    // Event "Pumpcellars_MiddlePumpcellar_Mode_c_off".
    IF NOT progress THEN
        b2 := (state0.dvar_M_Pumpcellars_MiddlePumpcellar_Mode) = (elit_drain);
        b2 := b2 OR ((state0.dvar_M_Pumpcellars_MiddlePumpcellar_Mode) = (elit_store));
        b1 := b2;
        b1 := b1 AND ((state0.dvar_M_RequirementStateEvtExcls) = (elit_X));
        IF b1 THEN
            b2 := (state0.dvar_M_Pumpcellars_MiddlePumpcellar_Control_Observer) = (elit_unpressed);
            IF NOT(b2) THEN
                b3 := (state0.dvar_M_Pumpcellars_MiddlePumpcellar_Control_Mode) = (elit_manual);
                b3 := b3 AND ((state0.dvar_M_Pumpcellars_MiddlePumpcellar_Control_Observer) <> (elit_autoPressed));
                b2 := b2 OR (b3);
            END_IF;
            b1 := b1 AND (b2);
        END_IF;
        b1 := b1 AND ((state0.dvar_M_Pumpcellars_MiddlePumpcellar_Control_Mode) = (elit_manual));
        b1 := b1 AND ((state0.dvar_M_Pumpcellars_MiddlePumpcellar_Control_Observer) = (elit_offPressed));
        b1 := b1 AND ((state0.dvar_M_Mutex1Home_TokenTracker) = (elit_Home));
        b1 := b1 AND ((state0.dvar_M_Mutex2Home_TokenTracker) = (elit_Home));
        b1 := b1 AND ((state0.dvar_M_sup1a) = (elit_X));
        b1 := b1 AND ((state0.dvar_M_sup2) = (elit_X));
        b1 := b1 AND ((state0.dvar_M_sup4) = (elit_X));
        IF b1 THEN
            progress := TRUE;
            state1 := state0;

            IF ((state0.dvar_M_HWMPCMode) = (elit_drain)) THEN
                state1.dvar_M_HWMPCMode_DRAIN := FALSE;
                state1.dvar_M_HWMPCMode_STORE := FALSE;
                state1.dvar_M_HWMPCMode_OFF := TRUE;
                state1.dvar_M_HWMPCMode := elit_off;
            ELSIF ((state0.dvar_M_HWMPCMode) = (elit_store)) THEN
                state1.dvar_M_HWMPCMode_DRAIN := FALSE;
                state1.dvar_M_HWMPCMode_STORE := FALSE;
                state1.dvar_M_HWMPCMode_OFF := TRUE;
                state1.dvar_M_HWMPCMode := elit_off;
            ELSIF ((state0.dvar_M_HWMPCMode) = (elit_off)) THEN
                state1.dvar_M_HWMPCMode := elit_off;
            END_IF;
            IF ((state0.dvar_M_Pumpcellars_MiddlePumpcellar_Mode) = (elit_drain)) THEN
                state1.dvar_M_Pumpcellars_MiddlePumpcellar_Mode := elit_off;
            ELSIF ((state0.dvar_M_Pumpcellars_MiddlePumpcellar_Mode) = (elit_store)) THEN
                state1.dvar_M_Pumpcellars_MiddlePumpcellar_Mode := elit_off;
            END_IF;

            state0 := state1;
        END_IF;
    END_IF;

    // Event "Pumpcellars_MiddlePumpcellar_Mode_c_store".
    IF NOT progress THEN
        b2 := (state0.dvar_M_Pumpcellars_MiddlePumpcellar_Mode) = (elit_drain);
        b2 := b2 OR ((state0.dvar_M_Pumpcellars_MiddlePumpcellar_Mode) = (elit_off));
        b1 := b2;
        b1 := b1 AND ((state0.dvar_M_RequirementStateEvtExcls) = (elit_X));
        IF b1 THEN
            b2 := (state0.dvar_M_Pumpcellars_MiddlePumpcellar_Control_Observer) = (elit_unpressed);
            IF NOT(b2) THEN
                b3 := (state0.dvar_M_Pumpcellars_MiddlePumpcellar_Control_Mode) = (elit_manual);
                b3 := b3 AND ((state0.dvar_M_Pumpcellars_MiddlePumpcellar_Control_Observer) <> (elit_autoPressed));
                b2 := b2 OR (b3);
            END_IF;
            b1 := b1 AND (b2);
        END_IF;
        IF b1 THEN
            b3 := (state0.dvar_M_Pumpcellars_MiddlePumpcellar_Control_Mode) = (elit_auto);
            b3 := b3 AND (NOT(((state0.dvar_M_Pumpcellars_Traffictube1_ModeTraffictube_Observer) = (elit_operational)) AND ((state0.dvar_M_Pumpcellars_Traffictube2_ModeTraffictube_Observer) = (elit_operational))));
            b2 := b3;
            IF NOT(b2) THEN
                b3 := (state0.dvar_M_Pumpcellars_MiddlePumpcellar_Control_Mode) = (elit_manual);
                b3 := b3 AND ((state0.dvar_M_Pumpcellars_MiddlePumpcellar_Control_Observer) = (elit_storePressed));
                b2 := b2 OR (b3);
            END_IF;
            b1 := b1 AND (b2);
        END_IF;
        b1 := b1 AND ((state0.dvar_M_Mutex1Home_TokenTracker) = (elit_Home));
        b1 := b1 AND ((state0.dvar_M_Mutex2Home_TokenTracker) = (elit_Home));
        b1 := b1 AND ((state0.dvar_M_sup1a) = (elit_X));
        b1 := b1 AND ((state0.dvar_M_sup2) = (elit_X));
        b1 := b1 AND ((state0.dvar_M_sup4) = (elit_X));
        IF b1 THEN
            progress := TRUE;
            state1 := state0;

            IF ((state0.dvar_M_HWMPCMode) = (elit_drain)) THEN
                state1.dvar_M_HWMPCMode_DRAIN := FALSE;
                state1.dvar_M_HWMPCMode_STORE := TRUE;
                state1.dvar_M_HWMPCMode_OFF := FALSE;
                state1.dvar_M_HWMPCMode := elit_store;
            ELSIF ((state0.dvar_M_HWMPCMode) = (elit_store)) THEN
                state1.dvar_M_HWMPCMode := elit_store;
            ELSIF ((state0.dvar_M_HWMPCMode) = (elit_off)) THEN
                state1.dvar_M_HWMPCMode_DRAIN := FALSE;
                state1.dvar_M_HWMPCMode_STORE := TRUE;
                state1.dvar_M_HWMPCMode_OFF := FALSE;
                state1.dvar_M_HWMPCMode := elit_store;
            END_IF;
            IF ((state0.dvar_M_Pumpcellars_MiddlePumpcellar_Mode) = (elit_drain)) THEN
                state1.dvar_M_Pumpcellars_MiddlePumpcellar_Mode := elit_store;
            ELSIF ((state0.dvar_M_Pumpcellars_MiddlePumpcellar_Mode) = (elit_off)) THEN
                state1.dvar_M_Pumpcellars_MiddlePumpcellar_Mode := elit_store;
            END_IF;

            state0 := state1;
        END_IF;
    END_IF;

    // Event "Pumpcellars_MiddlePumpcellar_PompRichting_c_hoofdPumpcellars1".
    IF NOT progress THEN
        IF (state0.dvar_M_MPC_HWPomprichting) = (elit_X) THEN
            progress := TRUE;
            state1 := state0;

            state1.dvar_M_MPC_HWPomprichting_HPC1 := TRUE;

            state0 := state1;
        END_IF;
    END_IF;

    // Event "Pumpcellars_MiddlePumpcellar_PompRichting_c_hoofdPumpcellars2".
    IF NOT progress THEN
        IF (state0.dvar_M_MPC_HWPomprichting) = (elit_X) THEN
            progress := TRUE;
            state1 := state0;

            state1.dvar_M_MPC_HWPomprichting_HPC1 := FALSE;

            state0 := state1;
        END_IF;
    END_IF;

    // Event "Pumpcellars_MiddlePumpcellar_Pump1_c_off".
    IF NOT progress THEN
        b1 := (state0.dvar_M_MPC_HWPump1) = (elit_X);
        b1 := b1 AND ((state0.dvar_M_Pumpcellars_MiddlePumpcellar_Pump1) = (elit_on));
        b1 := b1 AND ((state0.dvar_M_RequirementStateEvtExcls) = (elit_X));
        IF b1 THEN
            b3 := (state0.dvar_M_Pumpcellars_MiddlePumpcellar_Mode) = (elit_store);
            IF b3 THEN
                b4 := (state0.dvar_M_Pumpcellars_MiddlePumpcellar_SensorTank) = (elit_S2);
                b4 := b4 OR ((state0.dvar_M_Pumpcellars_MiddlePumpcellar_SensorTank) = (elit_S3));
                b4 := b4 OR ((state0.dvar_M_Pumpcellars_MiddlePumpcellar_SensorTank) = (elit_S1));
                b4 := b4 OR ((state0.dvar_M_Pumpcellars_MiddlePumpcellar_SensorTank) = (elit_Empty));
                b3 := b3 AND (b4);
            END_IF;
            b2 := b3;
            IF NOT(b2) THEN
                b3 := (state0.dvar_M_Pumpcellars_MiddlePumpcellar_Mode) = (elit_drain);
                b3 := b3 AND ((state0.dvar_M_Pumpcellars_MiddlePumpcellar_SensorTank) = (elit_Empty));
                b2 := b2 OR (b3);
            END_IF;
            b2 := b2 OR ((state0.dvar_M_Pumpcellars_MiddlePumpcellar_Mode) = (elit_off));
            b1 := b1 AND (b2);
        END_IF;
        b1 := b1 AND ((state0.dvar_M_Pumpcellars_MiddlePumpcellar_Control_Observer) = (elit_unpressed));
        b1 := b1 AND ((state0.dvar_M_sup2) = (elit_X));
        IF b1 THEN
            progress := TRUE;
            state1 := state0;

            state1.dvar_M_MPC_HWPump1_ON := FALSE;
            state1.dvar_M_Pumpcellars_MiddlePumpcellar_Pump1 := elit_off;

            state0 := state1;
        END_IF;
    END_IF;

    // Event "Pumpcellars_MiddlePumpcellar_Pump1_c_on".
    IF NOT progress THEN
        b1 := (state0.dvar_M_MPC_HWPump1) = (elit_X);
        b1 := b1 AND ((state0.dvar_M_Pumpcellars_MiddlePumpcellar_Pump1) = (elit_off));
        b1 := b1 AND ((state0.dvar_M_RequirementStateEvtExcls) = (elit_X));
        IF b1 THEN
            b3 := (state0.dvar_M_Pumpcellars_MiddlePumpcellar_Mode) = (elit_store);
            b3 := b3 AND ((state0.dvar_M_Pumpcellars_MiddlePumpcellar_SensorTank) = (elit_S5));
            b2 := b3;
            IF NOT(b2) THEN
                b3 := (state0.dvar_M_Pumpcellars_MiddlePumpcellar_Mode) = (elit_drain);
                IF b3 THEN
                    b4 := (state0.dvar_M_Pumpcellars_MiddlePumpcellar_SensorTank) = (elit_S2);
                    b4 := b4 OR ((state0.dvar_M_Pumpcellars_MiddlePumpcellar_SensorTank) = (elit_S3));
                    b4 := b4 OR ((state0.dvar_M_Pumpcellars_MiddlePumpcellar_SensorTank) = (elit_S4));
                    b4 := b4 OR ((state0.dvar_M_Pumpcellars_MiddlePumpcellar_SensorTank) = (elit_S5));
                    b3 := b3 AND (b4);
                END_IF;
                b2 := b2 OR (b3);
            END_IF;
            b1 := b1 AND (b2);
        END_IF;
        b1 := b1 AND ((state0.dvar_M_Pumpcellars_MiddlePumpcellar_Control_Observer) = (elit_unpressed));
        b1 := b1 AND ((state0.dvar_M_sup2) = (elit_X));
        IF b1 THEN
            progress := TRUE;
            state1 := state0;

            state1.dvar_M_MPC_HWPump1_ON := TRUE;
            state1.dvar_M_Pumpcellars_MiddlePumpcellar_Pump1 := elit_on;

            state0 := state1;
        END_IF;
    END_IF;

    // Event "Pumpcellars_MiddlePumpcellar_Pump2_c_off".
    IF NOT progress THEN
        b1 := (state0.dvar_M_MPC_HWPump2) = (elit_X);
        b1 := b1 AND ((state0.dvar_M_Pumpcellars_MiddlePumpcellar_Pump2) = (elit_on));
        b1 := b1 AND ((state0.dvar_M_RequirementStateEvtExcls) = (elit_X));
        IF b1 THEN
            b3 := (state0.dvar_M_Pumpcellars_MiddlePumpcellar_Mode) = (elit_store);
            IF b3 THEN
                b4 := (state0.dvar_M_Pumpcellars_MiddlePumpcellar_SensorTank) = (elit_S2);
                b4 := b4 OR ((state0.dvar_M_Pumpcellars_MiddlePumpcellar_SensorTank) = (elit_S3));
                b4 := b4 OR ((state0.dvar_M_Pumpcellars_MiddlePumpcellar_SensorTank) = (elit_S1));
                b4 := b4 OR ((state0.dvar_M_Pumpcellars_MiddlePumpcellar_SensorTank) = (elit_Empty));
                b3 := b3 AND (b4);
            END_IF;
            b2 := b3;
            IF NOT(b2) THEN
                b3 := (state0.dvar_M_Pumpcellars_MiddlePumpcellar_Mode) = (elit_drain);
                b3 := b3 AND ((state0.dvar_M_Pumpcellars_MiddlePumpcellar_SensorTank) = (elit_Empty));
                b2 := b2 OR (b3);
            END_IF;
            b2 := b2 OR ((state0.dvar_M_Pumpcellars_MiddlePumpcellar_Mode) = (elit_off));
            b1 := b1 AND (b2);
        END_IF;
        b1 := b1 AND ((state0.dvar_M_Pumpcellars_MiddlePumpcellar_Control_Observer) = (elit_unpressed));
        b1 := b1 AND ((state0.dvar_M_sup2) = (elit_X));
        IF b1 THEN
            progress := TRUE;
            state1 := state0;

            state1.dvar_M_MPC_HWPump2_ON := FALSE;
            state1.dvar_M_Pumpcellars_MiddlePumpcellar_Pump2 := elit_off;

            state0 := state1;
        END_IF;
    END_IF;

    // Event "Pumpcellars_MiddlePumpcellar_Pump2_c_on".
    IF NOT progress THEN
        b1 := (state0.dvar_M_MPC_HWPump2) = (elit_X);
        b1 := b1 AND ((state0.dvar_M_Pumpcellars_MiddlePumpcellar_Pump2) = (elit_off));
        b1 := b1 AND ((state0.dvar_M_RequirementStateEvtExcls) = (elit_X));
        IF b1 THEN
            b3 := (state0.dvar_M_Pumpcellars_MiddlePumpcellar_Mode) = (elit_store);
            b3 := b3 AND ((state0.dvar_M_Pumpcellars_MiddlePumpcellar_SensorTank) = (elit_S5));
            b2 := b3;
            IF NOT(b2) THEN
                b3 := (state0.dvar_M_Pumpcellars_MiddlePumpcellar_Mode) = (elit_drain);
                IF b3 THEN
                    b4 := (state0.dvar_M_Pumpcellars_MiddlePumpcellar_SensorTank) = (elit_S3);
                    b4 := b4 OR ((state0.dvar_M_Pumpcellars_MiddlePumpcellar_SensorTank) = (elit_S4));
                    b4 := b4 OR ((state0.dvar_M_Pumpcellars_MiddlePumpcellar_SensorTank) = (elit_S5));
                    b3 := b3 AND (b4);
                END_IF;
                b2 := b2 OR (b3);
            END_IF;
            b1 := b1 AND (b2);
        END_IF;
        b1 := b1 AND ((state0.dvar_M_Pumpcellars_MiddlePumpcellar_Control_Observer) = (elit_unpressed));
        b1 := b1 AND ((state0.dvar_M_sup2) = (elit_X));
        IF b1 THEN
            progress := TRUE;
            state1 := state0;

            state1.dvar_M_MPC_HWPump2_ON := TRUE;
            state1.dvar_M_Pumpcellars_MiddlePumpcellar_Pump2 := elit_on;

            state0 := state1;
        END_IF;
    END_IF;

    // Event "Pumpcellars_MiddlePumpcellar_PumpDirection_c_headPumpcellar1".
    IF NOT progress THEN
        b1 := (state0.dvar_M_Pumpcellars_MiddlePumpcellar_PumpDirection) = (elit_headPumpcellar2);
        b1 := b1 AND ((state0.dvar_M_RequirementStateEvtExcls) = (elit_X));
        b1 := b1 AND ((state0.dvar_M_Pumpcellars_HeadPumpcellar1_SensorTank) = (elit_S4));
        b1 := b1 AND ((state0.dvar_M_sup5) = (elit_X));
        IF b1 THEN
            progress := TRUE;
            state1 := state0;

            state1.dvar_M_Pumpcellars_MiddlePumpcellar_PumpDirection := elit_headPumpcellar1;

            state0 := state1;
        END_IF;
    END_IF;

    // Event "Pumpcellars_MiddlePumpcellar_PumpDirection_c_headPumpcellar2".
    IF NOT progress THEN
        b1 := (state0.dvar_M_Pumpcellars_MiddlePumpcellar_PumpDirection) = (elit_headPumpcellar1);
        b1 := b1 AND ((state0.dvar_M_RequirementStateEvtExcls) = (elit_X));
        b1 := b1 AND ((state0.dvar_M_Pumpcellars_HeadPumpcellar1_SensorTank) = (elit_S5));
        b1 := b1 AND ((state0.dvar_M_sup5) = (elit_X));
        IF b1 THEN
            progress := TRUE;
            state1 := state0;

            state1.dvar_M_Pumpcellars_MiddlePumpcellar_PumpDirection := elit_headPumpcellar2;

            state0 := state1;
        END_IF;
    END_IF;

    // Event "Pumpcellars_MiddlePumpcellar_SensorTank_u_S1off".
    IF NOT progress THEN
        b1 := (state0.dvar_M_MPC_HWSensorS1) = (elit_on);
        b1 := b1 AND (NOT(ivar_M_MPC_HWSensorS1_ON));
        b1 := b1 AND ((state0.dvar_M_Pumpcellars_MiddlePumpcellar_SensorTank) = (elit_S1));
        IF b1 THEN
            b2 := (state0.dvar_M_Pumpcellars_MiddlePumpcellar_Pump1) = (elit_on);
            b2 := b2 OR ((state0.dvar_M_Pumpcellars_MiddlePumpcellar_Pump2) = (elit_on));
            b1 := b1 AND (b2);
        END_IF;
        IF b1 THEN
            progress := TRUE;
            state1 := state0;

            state1.dvar_M_MPC_HWSensorS1 := elit_off;
            state1.dvar_M_Pumpcellars_MiddlePumpcellar_SensorTank := elit_Empty;

            state0 := state1;
        END_IF;
    END_IF;

    // Event "Pumpcellars_MiddlePumpcellar_SensorTank_u_S1on".
    IF NOT progress THEN
        b1 := (state0.dvar_M_MPC_HWSensorS1) = (elit_off);
        b1 := b1 AND (ivar_M_MPC_HWSensorS1_ON);
        b1 := b1 AND ((state0.dvar_M_Pumpcellars_MiddlePumpcellar_SensorTank) = (elit_Empty));
        IF b1 THEN
            progress := TRUE;
            state1 := state0;

            state1.dvar_M_MPC_HWSensorS1 := elit_on;
            state1.dvar_M_Pumpcellars_MiddlePumpcellar_SensorTank := elit_S1;

            state0 := state1;
        END_IF;
    END_IF;

    // Event "Pumpcellars_MiddlePumpcellar_SensorTank_u_S2off".
    IF NOT progress THEN
        b1 := (state0.dvar_M_MPC_HWSensorS2) = (elit_on);
        b1 := b1 AND (NOT(ivar_M_MPC_HWSensorS2_ON));
        b1 := b1 AND ((state0.dvar_M_Pumpcellars_MiddlePumpcellar_SensorTank) = (elit_S2));
        IF b1 THEN
            b2 := (state0.dvar_M_Pumpcellars_MiddlePumpcellar_Pump1) = (elit_on);
            b2 := b2 OR ((state0.dvar_M_Pumpcellars_MiddlePumpcellar_Pump2) = (elit_on));
            b1 := b1 AND (b2);
        END_IF;
        IF b1 THEN
            progress := TRUE;
            state1 := state0;

            state1.dvar_M_MPC_HWSensorS2 := elit_off;
            state1.dvar_M_Pumpcellars_MiddlePumpcellar_SensorTank := elit_S1;

            state0 := state1;
        END_IF;
    END_IF;

    // Event "Pumpcellars_MiddlePumpcellar_SensorTank_u_S2on".
    IF NOT progress THEN
        b1 := (state0.dvar_M_MPC_HWSensorS2) = (elit_off);
        b1 := b1 AND (ivar_M_MPC_HWSensorS2_ON);
        b1 := b1 AND ((state0.dvar_M_Pumpcellars_MiddlePumpcellar_SensorTank) = (elit_S1));
        IF b1 THEN
            progress := TRUE;
            state1 := state0;

            state1.dvar_M_MPC_HWSensorS2 := elit_on;
            state1.dvar_M_Pumpcellars_MiddlePumpcellar_SensorTank := elit_S2;

            state0 := state1;
        END_IF;
    END_IF;

    // Event "Pumpcellars_MiddlePumpcellar_SensorTank_u_S3off".
    IF NOT progress THEN
        b1 := (state0.dvar_M_MPC_HWSensorS3) = (elit_on);
        b1 := b1 AND (NOT(ivar_M_MPC_HWSensorS3_ON));
        b1 := b1 AND ((state0.dvar_M_Pumpcellars_MiddlePumpcellar_SensorTank) = (elit_S3));
        IF b1 THEN
            b2 := (state0.dvar_M_Pumpcellars_MiddlePumpcellar_Pump1) = (elit_on);
            b2 := b2 OR ((state0.dvar_M_Pumpcellars_MiddlePumpcellar_Pump2) = (elit_on));
            b1 := b1 AND (b2);
        END_IF;
        IF b1 THEN
            progress := TRUE;
            state1 := state0;

            state1.dvar_M_MPC_HWSensorS3 := elit_off;
            state1.dvar_M_Pumpcellars_MiddlePumpcellar_SensorTank := elit_S2;

            state0 := state1;
        END_IF;
    END_IF;

    // Event "Pumpcellars_MiddlePumpcellar_SensorTank_u_S3on".
    IF NOT progress THEN
        b1 := (state0.dvar_M_MPC_HWSensorS3) = (elit_off);
        b1 := b1 AND (ivar_M_MPC_HWSensorS3_ON);
        b1 := b1 AND ((state0.dvar_M_Pumpcellars_MiddlePumpcellar_SensorTank) = (elit_S2));
        IF b1 THEN
            progress := TRUE;
            state1 := state0;

            state1.dvar_M_MPC_HWSensorS3 := elit_on;
            state1.dvar_M_Pumpcellars_MiddlePumpcellar_SensorTank := elit_S3;

            state0 := state1;
        END_IF;
    END_IF;

    // Event "Pumpcellars_MiddlePumpcellar_SensorTank_u_S4off".
    IF NOT progress THEN
        b1 := (state0.dvar_M_MPC_HWSensorS4) = (elit_on);
        b1 := b1 AND (NOT(ivar_M_MPC_HWSensorS4_ON));
        b1 := b1 AND ((state0.dvar_M_Pumpcellars_MiddlePumpcellar_SensorTank) = (elit_S4));
        IF b1 THEN
            b2 := (state0.dvar_M_Pumpcellars_MiddlePumpcellar_Pump1) = (elit_on);
            b2 := b2 OR ((state0.dvar_M_Pumpcellars_MiddlePumpcellar_Pump2) = (elit_on));
            b1 := b1 AND (b2);
        END_IF;
        IF b1 THEN
            progress := TRUE;
            state1 := state0;

            state1.dvar_M_MPC_HWSensorS4 := elit_off;
            state1.dvar_M_Pumpcellars_MiddlePumpcellar_SensorTank := elit_S3;

            state0 := state1;
        END_IF;
    END_IF;

    // Event "Pumpcellars_MiddlePumpcellar_SensorTank_u_S4on".
    IF NOT progress THEN
        b1 := (state0.dvar_M_MPC_HWSensorS4) = (elit_off);
        b1 := b1 AND (ivar_M_MPC_HWSensorS4_ON);
        b1 := b1 AND ((state0.dvar_M_Pumpcellars_MiddlePumpcellar_SensorTank) = (elit_S3));
        IF b1 THEN
            progress := TRUE;
            state1 := state0;

            state1.dvar_M_MPC_HWSensorS4 := elit_on;
            state1.dvar_M_Pumpcellars_MiddlePumpcellar_SensorTank := elit_S4;

            state0 := state1;
        END_IF;
    END_IF;

    // Event "Pumpcellars_MiddlePumpcellar_SensorTank_u_S5off".
    IF NOT progress THEN
        b1 := (state0.dvar_M_MPC_HWSensorS5) = (elit_on);
        b1 := b1 AND (NOT(ivar_M_MPC_HWSensorS5_ON));
        b1 := b1 AND ((state0.dvar_M_Pumpcellars_MiddlePumpcellar_SensorTank) = (elit_S5));
        IF b1 THEN
            b2 := (state0.dvar_M_Pumpcellars_MiddlePumpcellar_Pump1) = (elit_on);
            b2 := b2 OR ((state0.dvar_M_Pumpcellars_MiddlePumpcellar_Pump2) = (elit_on));
            b1 := b1 AND (b2);
        END_IF;
        IF b1 THEN
            progress := TRUE;
            state1 := state0;

            state1.dvar_M_MPC_HWSensorS5 := elit_off;
            state1.dvar_M_Pumpcellars_MiddlePumpcellar_SensorTank := elit_S4;

            state0 := state1;
        END_IF;
    END_IF;

    // Event "Pumpcellars_MiddlePumpcellar_SensorTank_u_S5on".
    IF NOT progress THEN
        b1 := (state0.dvar_M_MPC_HWSensorS5) = (elit_off);
        b1 := b1 AND (ivar_M_MPC_HWSensorS5_ON);
        b1 := b1 AND ((state0.dvar_M_Pumpcellars_MiddlePumpcellar_SensorTank) = (elit_S4));
        IF b1 THEN
            progress := TRUE;
            state1 := state0;

            state1.dvar_M_MPC_HWSensorS5 := elit_on;
            state1.dvar_M_Pumpcellars_MiddlePumpcellar_SensorTank := elit_S5;

            state0 := state1;
        END_IF;
    END_IF;

    // Event "Pumpcellars_Traffictube1_Observer_c_emergency".
    IF NOT progress THEN
        b1 := (state0.dvar_M_HWModeTraffictube1Observer) = (elit_X);
        b1 := b1 AND (ivar_TT1EMERGENCY);
        b1 := b1 AND (NOT(ivar_TT1OPERATIONAL));
        b1 := b1 AND (NOT(ivar_TT1RECOVERY));
        IF b1 THEN
            b2 := (state0.dvar_M_Pumpcellars_Traffictube1_ModeTraffictube_Observer) = (elit_operational);
            b2 := b2 OR ((state0.dvar_M_Pumpcellars_Traffictube1_ModeTraffictube_Observer) = (elit_recovery));
            b1 := b1 AND (b2);
        END_IF;
        IF b1 THEN
            progress := TRUE;
            state1 := state0;

            IF ((state0.dvar_M_Pumpcellars_Traffictube1_ModeTraffictube_Observer) = (elit_operational)) THEN
                state1.dvar_M_Pumpcellars_Traffictube1_ModeTraffictube_Observer := elit_emergency;
            ELSIF ((state0.dvar_M_Pumpcellars_Traffictube1_ModeTraffictube_Observer) = (elit_recovery)) THEN
                state1.dvar_M_Pumpcellars_Traffictube1_ModeTraffictube_Observer := elit_emergency;
            END_IF;

            state0 := state1;
        END_IF;
    END_IF;

    // Event "Pumpcellars_Traffictube1_Observer_c_operational".
    IF NOT progress THEN
        b1 := (state0.dvar_M_HWModeTraffictube1Observer) = (elit_X);
        b1 := b1 AND (NOT(ivar_TT1EMERGENCY));
        b1 := b1 AND (ivar_TT1OPERATIONAL);
        b1 := b1 AND (NOT(ivar_TT1RECOVERY));
        IF b1 THEN
            b2 := (state0.dvar_M_Pumpcellars_Traffictube1_ModeTraffictube_Observer) = (elit_emergency);
            b2 := b2 OR ((state0.dvar_M_Pumpcellars_Traffictube1_ModeTraffictube_Observer) = (elit_recovery));
            b1 := b1 AND (b2);
        END_IF;
        IF b1 THEN
            progress := TRUE;
            state1 := state0;

            IF ((state0.dvar_M_Pumpcellars_Traffictube1_ModeTraffictube_Observer) = (elit_emergency)) THEN
                state1.dvar_M_Pumpcellars_Traffictube1_ModeTraffictube_Observer := elit_operational;
            ELSIF ((state0.dvar_M_Pumpcellars_Traffictube1_ModeTraffictube_Observer) = (elit_recovery)) THEN
                state1.dvar_M_Pumpcellars_Traffictube1_ModeTraffictube_Observer := elit_operational;
            END_IF;

            state0 := state1;
        END_IF;
    END_IF;

    // Event "Pumpcellars_Traffictube1_Observer_c_recovery".
    IF NOT progress THEN
        b1 := (state0.dvar_M_HWModeTraffictube1Observer) = (elit_X);
        b1 := b1 AND (NOT(ivar_TT1EMERGENCY));
        b1 := b1 AND (NOT(ivar_TT1OPERATIONAL));
        b1 := b1 AND (ivar_TT1RECOVERY);
        IF b1 THEN
            b2 := (state0.dvar_M_Pumpcellars_Traffictube1_ModeTraffictube_Observer) = (elit_operational);
            b2 := b2 OR ((state0.dvar_M_Pumpcellars_Traffictube1_ModeTraffictube_Observer) = (elit_emergency));
            b1 := b1 AND (b2);
        END_IF;
        IF b1 THEN
            progress := TRUE;
            state1 := state0;

            IF ((state0.dvar_M_Pumpcellars_Traffictube1_ModeTraffictube_Observer) = (elit_operational)) THEN
                state1.dvar_M_Pumpcellars_Traffictube1_ModeTraffictube_Observer := elit_recovery;
            ELSIF ((state0.dvar_M_Pumpcellars_Traffictube1_ModeTraffictube_Observer) = (elit_emergency)) THEN
                state1.dvar_M_Pumpcellars_Traffictube1_ModeTraffictube_Observer := elit_recovery;
            END_IF;

            state0 := state1;
        END_IF;
    END_IF;

    // Event "Pumpcellars_Traffictube2_Observer_c_emergency".
    IF NOT progress THEN
        b1 := (state0.dvar_M_HWModeTraffictube2Observer) = (elit_X);
        b1 := b1 AND (ivar_TT2EMERGENCY);
        b1 := b1 AND (NOT(ivar_TT2OPERATIONAL));
        b1 := b1 AND (NOT(ivar_TT2RECOVERY));
        IF b1 THEN
            b2 := (state0.dvar_M_Pumpcellars_Traffictube2_ModeTraffictube_Observer) = (elit_operational);
            b2 := b2 OR ((state0.dvar_M_Pumpcellars_Traffictube2_ModeTraffictube_Observer) = (elit_recovery));
            b1 := b1 AND (b2);
        END_IF;
        IF b1 THEN
            progress := TRUE;
            state1 := state0;

            IF ((state0.dvar_M_Pumpcellars_Traffictube2_ModeTraffictube_Observer) = (elit_operational)) THEN
                state1.dvar_M_Pumpcellars_Traffictube2_ModeTraffictube_Observer := elit_emergency;
            ELSIF ((state0.dvar_M_Pumpcellars_Traffictube2_ModeTraffictube_Observer) = (elit_recovery)) THEN
                state1.dvar_M_Pumpcellars_Traffictube2_ModeTraffictube_Observer := elit_emergency;
            END_IF;

            state0 := state1;
        END_IF;
    END_IF;

    // Event "Pumpcellars_Traffictube2_Observer_c_operational".
    IF NOT progress THEN
        b1 := (state0.dvar_M_HWModeTraffictube2Observer) = (elit_X);
        b1 := b1 AND (NOT(ivar_TT2EMERGENCY));
        b1 := b1 AND (ivar_TT2OPERATIONAL);
        b1 := b1 AND (NOT(ivar_TT2RECOVERY));
        IF b1 THEN
            b2 := (state0.dvar_M_Pumpcellars_Traffictube2_ModeTraffictube_Observer) = (elit_emergency);
            b2 := b2 OR ((state0.dvar_M_Pumpcellars_Traffictube2_ModeTraffictube_Observer) = (elit_recovery));
            b1 := b1 AND (b2);
        END_IF;
        IF b1 THEN
            progress := TRUE;
            state1 := state0;

            IF ((state0.dvar_M_Pumpcellars_Traffictube2_ModeTraffictube_Observer) = (elit_emergency)) THEN
                state1.dvar_M_Pumpcellars_Traffictube2_ModeTraffictube_Observer := elit_operational;
            ELSIF ((state0.dvar_M_Pumpcellars_Traffictube2_ModeTraffictube_Observer) = (elit_recovery)) THEN
                state1.dvar_M_Pumpcellars_Traffictube2_ModeTraffictube_Observer := elit_operational;
            END_IF;

            state0 := state1;
        END_IF;
    END_IF;

    // Event "Pumpcellars_Traffictube2_Observer_c_recovery".
    IF NOT progress THEN
        b1 := (state0.dvar_M_HWModeTraffictube2Observer) = (elit_X);
        b1 := b1 AND (NOT(ivar_TT2EMERGENCY));
        b1 := b1 AND (NOT(ivar_TT2OPERATIONAL));
        b1 := b1 AND (ivar_TT2RECOVERY);
        IF b1 THEN
            b2 := (state0.dvar_M_Pumpcellars_Traffictube2_ModeTraffictube_Observer) = (elit_operational);
            b2 := b2 OR ((state0.dvar_M_Pumpcellars_Traffictube2_ModeTraffictube_Observer) = (elit_emergency));
            b1 := b1 AND (b2);
        END_IF;
        IF b1 THEN
            progress := TRUE;
            state1 := state0;

            IF ((state0.dvar_M_Pumpcellars_Traffictube2_ModeTraffictube_Observer) = (elit_operational)) THEN
                state1.dvar_M_Pumpcellars_Traffictube2_ModeTraffictube_Observer := elit_recovery;
            ELSIF ((state0.dvar_M_Pumpcellars_Traffictube2_ModeTraffictube_Observer) = (elit_emergency)) THEN
                state1.dvar_M_Pumpcellars_Traffictube2_ModeTraffictube_Observer := elit_recovery;
            END_IF;

            state0 := state1;
        END_IF;
    END_IF;

    // Done with events?
    IF NOT progress THEN
        EXIT;
    END_IF;

    // Protect against events that are always enabled.
    loopCount := loopCount + 1;
    IF loopCount >= 100 THEN
        loopsKilled := loopsKilled + 1;
        EXIT;
    END_IF;
END_WHILE;
          
END_PROGRAM

CONFIGURATION config
  RESOURCE Untitled1 ON PLC
    VAR_GLOBAL  (* INPUTS *)
      ivar_Mutex1Home_R2 AT %I* : BOOL;
      ivar_Mutex2Home_R2 AT %I* : BOOL;
      ivar_Mutex3Home_R2 AT %I* : BOOL;
      ivar_Mutex4Home_R2 AT %I* : BOOL;
      ivar_TT1EMERGENCY AT %I* : BOOL;
      ivar_TT1RECOVERY AT %I* : BOOL;
      ivar_TT1OPERATIONAL AT %I* : BOOL;
      ivar_TT2EMERGENCY AT %I* : BOOL;
      ivar_TT2RECOVERY AT %I* : BOOL;
      ivar_TT2OPERATIONAL AT %I* : BOOL;
      ivar_M_HPC1_HWSensorS1_ON AT %I* : BOOL;
      ivar_M_HPC1_HWSensorS2_ON AT %I* : BOOL;
      ivar_M_HPC1_HWSensorS3_ON AT %I* : BOOL;
      ivar_M_HPC1_HWSensorS4_ON AT %I* : BOOL;
      ivar_M_HPC1_HWSensorS5_ON AT %I* : BOOL;
      ivar_M_HWHPC1ControlButtonAuto_PUSHED AT %I* : BOOL;
      ivar_M_HWHPC1ControlButtonManual_PUSHED AT %I* : BOOL;
      ivar_M_HWHPC1ModeButtonDrain_PUSHED AT %I* : BOOL;
      ivar_M_HWHPC1ModeButtonOff_PUSHED AT %I* : BOOL;
      ivar_M_HWHPC1ModeButtonStore_PUSHED AT %I* : BOOL;
      ivar_M_HWMPCControlButtonAuto_PUSHED AT %I* : BOOL;
      ivar_M_HWMPCControlButtonManual_PUSHED AT %I* : BOOL;
      ivar_M_HWMPCModeButtonDrain_PUSHED AT %I* : BOOL;
      ivar_M_HWMPCModeButtonOff_PUSHED AT %I* : BOOL;
      ivar_M_HWMPCModeButtonStore_PUSHED AT %I* : BOOL;
      ivar_M_HWMutex1_There AT %I* : BOOL;
      ivar_M_HWMutex1_SendingHere AT %I* : BOOL;
      ivar_M_HWMutex2_There AT %I* : BOOL;
      ivar_M_HWMutex2_SendingHere AT %I* : BOOL;
      ivar_M_HWMutex3_There AT %I* : BOOL;
      ivar_M_HWMutex3_SendingHere AT %I* : BOOL;
      ivar_M_HWMutex4_There AT %I* : BOOL;
      ivar_M_HWMutex4_SendingHere AT %I* : BOOL;
      ivar_M_MPC_HWSensorS1_ON AT %I* : BOOL;
      ivar_M_MPC_HWSensorS2_ON AT %I* : BOOL;
      ivar_M_MPC_HWSensorS3_ON AT %I* : BOOL;
      ivar_M_MPC_HWSensorS4_ON AT %I* : BOOL;
      ivar_M_MPC_HWSensorS5_ON AT %I* : BOOL;
    END_VAR
    VAR_GLOBAL  (* TIMERS *)
      timer0 : TON;
      timer1 : TON;
      curTimer : INT := 0;
    END_VAR
    TASK PlcTask(INTERVAL := t#10ms, PRIORITY := 20);
    PROGRAM MAIN WITH PlcTask : MAIN;
  END_RESOURCE
END_CONFIGURATION
